PROGRAM P_Demo_LTIME_TO_PMLTime
VAR
    tInput          : LTIME := LTIME#1H30M;       // 演示用：1 小时 30 分钟时长
    stPMLDuration   : ST_PMLDateAndTime;          // 转换结果（在线观察各字段）
END_VAR

// ============================================================
// Tc3_PackML_V3.LTIME_TO_PMLTime 演示程序
// ============================================================
// 场景：把 LTIME 类型的累计运行时长转成 PackML ST_PMLDateAndTime 结构体
//       写入 Admin PackTag 时间字段。
// 价值：标准化 LTIME → PackML 时长结构转换，避免手写时长拆解。V3 用结构体
//       返回（V2 用数组）：字段名访问更安全、可读性更好。
// 验证：登录后看 stPMLDuration.Hour 字段：tInput=LTIME#1H30M 应得
//       Hour=1, Minute=30, 其余字段为 0。
// 验证步骤：
//   1. 右键 PLC 项目下 POUs 文件夹 → Add → Existing Item → 选本 .TcPOU 文件
//   2. 引用 Tc3_PackML_V3（References → Add library）
//   3. 编译 → 登录 → 运行；按上方"验证"指引在线写值观察
// ============================================================

(* 纯函数调用——单行完成 *)
stPMLDuration := LTIME_TO_PMLTime(Input := tInput);

END_PROGRAM

(* stored: Version 1.1.0.1, ProductVersion 3.1.4024.5
   POU P_Demo_LTIME_TO_PMLTime: Id {f4cc2184-f703-5bf1-8448-a82329510ede}, SpecialFunc None *)
